FUNCTION_BLOCK IAS_SKILL_MUX_GEN (* Composite Function Block Type *)
  (* Standard: 61499-2 *)
  (* Version 0.0, 2008-07-10, 4DIAC-IDE, 4DIAC-Consortium *)
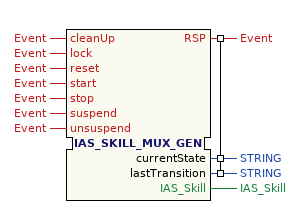
  EVENT_INPUT
    cleanUp;
    lock;
    reset;
    start;
    stop;
    suspend;
    unsuspend;
  END_EVENT
  EVENT_OUTPUT
    RSP WITH currentState, lastTransition;
  END_EVENT
  VAR_OUTPUT
    currentState : STRING;
    lastTransition : STRING;
  END_VAR
  PLUGS
    IAS_Skill : IAS_Skill;
  END_PLUGS
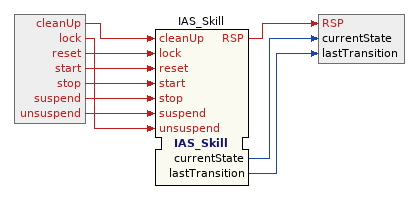
  EVENT_CONNECTIONS
    cleanUp TO IAS_Skill.cleanUp;
    lock TO IAS_Skill.lock;
    reset TO IAS_Skill.reset;
    start TO IAS_Skill.start;
    stop TO IAS_Skill.stop;
    suspend TO IAS_Skill.suspend;
    unsuspend TO IAS_Skill.unsuspend;
    IAS_Skill.RSP TO RSP;
  END_CONNECTIONS
  DATA_CONNECTIONS
    IAS_Skill.currentState TO currentState;
    IAS_Skill.lastTransition TO lastTransition;
  END_CONNECTIONS
END_FUNCTION_BLOCK
